// TIA Portal V20 export
FUNCTION_BLOCK "FB_WarmUP"   // FB530, SCL
{ S7_Optimized_Access := 'TRUE' }
// stored: AutoNumber false, MemoryReserve 100, SetENOAutomatically false
   VAR
      sWarmUpTimer : Time;
      sLimitedWarmupTime : Bool;
      sUnlimitedWarmupTime : Bool;
      sActualWarmupTime : Time;
      sRemainingWarmupMinutes : Int;
      sDeltaTimeWarmup : Time;
      sLimitedWarmUP : TON_TIME;
      sStartWarmup { S7_SetPoint := 'True'} : Bool;
      sUnlimitedWarmUP : TON_TIME;
      sUnlimitedWarmUPCounter { S7_SetPoint := 'True'} : "FB_TimeCounter";
   END_VAR
   VAR CONSTANT
      WU_MIN : Int := 30;
   END_VAR
BEGIN
   REGION Description header 
       //==================================================================================
       // POSALUX Swiss SA / (C) Copyright 2024
       //----------------------------------------------------------------------------------
       // Title: Laser Warm-up
       // Comment/Function: 
       // This block manages the laser warm-up process. It includes functionality for both limited
       // and unlimited warm-up times.
       //
       // Author: [Gowsigan SRITHARAN]
       // Engineering: TIA Portal [version]
       //----------------------------------------------------------------------------------
       // Change log table:
       // Version  | Date     | Expert in charge | Changes applied
       // ---------|----------|------------------|------------------------------------
       // 00.00.01 | 20250224 | gsr              | First released version
       // 00.00.02 | 20250314 | wfa              | Modification unlimited timer
       // ==================================================================================
   END_REGION

   REGION Selection Warm-UP mode: limited or unlimited
       // Timer for unlimited Warm-UP detection
       #sUnlimitedWarmUP(IN := "DB_McpKeyboardSignals".sK14_WarmUp.sKeySWStatus OR "DB_HmiKeyboardSignals".sK14_WarmUp.sKeySWStatus,
                         PT := T#2s);

       // Warm-up mode selection logic
       IF ("DB_McpKeyboardSignals".sK14_WarmUp.sKeySWStatus OR "DB_HmiKeyboardSignals".sK14_WarmUp.sKeySWStatus) AND "LBP_ModeGroup".E_AUTO AND NOT #sUnlimitedWarmUP.Q THEN
           // Activate unlimited Warm-UP when key is initially pressed
           #sLimitedWarmupTime := FALSE;
           #sUnlimitedWarmupTime := TRUE;
           #sStartWarmup := TRUE;
       ELSIF "DB_McpKeyboardSignals".sK14_WarmUp.sKeySWStatus AND "DB_HmiKeyboardSignals".sK14_WarmUp.sKeySWStatus AND "LBP_ModeGroup".E_AUTO AND #sUnlimitedWarmUP.Q THEN
           // Switch to limited Warm-UP if key is held for 2 seconds
           #sLimitedWarmupTime := TRUE;
           #sUnlimitedWarmupTime := FALSE;
           #sStartWarmup := TRUE;
           #sWarmUpTimer := DINT_TO_TIME(DINT_TO_INT(#WU_MIN * 60 * 1000)); // Limited time in milliseconds
       ELSIF "DB_McpKeyboardSignals".sK14_WarmUp.sKeySWToggleStatus = FALSE AND "DB_HmiKeyboardSignals".sK14_WarmUp.sKeySWToggleStatus THEN
           #sLimitedWarmupTime := FALSE;
           #sUnlimitedWarmupTime := FALSE;
           #sStartWarmup := FALSE;
       END_IF;
   END_REGION

   REGION Warm-UP Counter (Unlimited Warm-Up)
       #sUnlimitedWarmUPCounter(iStart := #sUnlimitedWarmupTime AND ("LBP_Chan1".E_ProgRunning OR "LBP_Chan1".E_ProgWait OR "LBP_Chan1".E_ProgStop),
                                iReset := NOT "DB_McpKeyboardSignals".sK14_WarmUp.sKeySWToggleStatus AND NOT "DB_HmiKeyboardSignals".sK14_WarmUp.sKeySWToggleStatus);
   END_REGION ;

   REGION Warm-UP Timer  (Limited Warm-up)  
       // Start the Warm-UP timer
       #sLimitedWarmUP.TON(IN := #sLimitedWarmupTime AND ("LBP_Chan1".E_ProgRunning OR "LBP_Chan1".E_ProgWait OR "LBP_Chan1".E_ProgStop),
                           PT := #sWarmUpTimer);

       IF #sLimitedWarmUP.Q THEN
           "DB_McpKeyboardSignals".sK14_WarmUp.sKeySWToggleStatus := FALSE;
           "DB_HmiKeyboardSignals".sK14_WarmUp.sKeySWToggleStatus := FALSE;
       END_IF;
   END_REGION

   REGION Update NC inputs and MCP LED status
       "LBP_NC".A_Set_Inp34 := "DB_McpKeyboardSignals".sK14_WarmUp.sKeySWToggleStatus OR "DB_HmiKeyboardSignals".sK14_WarmUp.sKeySWToggleStatus;

       "DB_McpKeyboardSignals".sK14_WarmUp.sLedSWStatus :=
       "DB_McpKeyboardSignals".sK14_WarmUp.sKeySWToggleStatus
       AND (#sUnlimitedWarmupTime OR "Clock_2Hz");

       "DB_HmiKeyboardSignals".sK14_WarmUp.sLedSWStatus :=
       "DB_HmiKeyboardSignals".sK14_WarmUp.sKeySWToggleStatus
       AND (#sUnlimitedWarmupTime OR "Clock_2Hz");
   END_REGION

   REGION Display Remaining Time
       IF #sLimitedWarmupTime THEN
           // Display remaining time for limited warm-up
           "DB_HMIStatus".WarmUpTime := DINT_TO_REAL(TIME_TO_DINT(#sLimitedWarmUP.PT - #sLimitedWarmUP.ET)) / 1000.0;
       ELSIF #sUnlimitedWarmupTime THEN
           // Display elapsed time for unlimited warm-up
           "DB_HMIStatus".WarmUpTime := #sUnlimitedWarmUPCounter.ioSecondsCumul;
       ELSE
           // Reset display when conditions are not met
           "DB_HMIStatus".WarmUpTime := 0;
       END_IF;
   END_REGION

   REGION Warm-UP Message
       IF "LBP_ModeGroup".E_AUTO AND "LBP_NC".A_Set_Inp34 AND
           ("LBP_Chan1".E_ProgRunning OR "LBP_Chan1".E_ProgWait OR "LBP_Chan1".E_ProgStop) THEN
           "LBP_AlarmMsgs".UserA[0].A70UUxx[35] := TRUE;
       END_IF;
   END_REGION

   REGION Warm-UP Status
       "DB_HMIStatus".WarmUpOn := #sStartWarmup;
   END_REGION

   REGION Warm-UP Status To NC
       "DB_PLC_ISO_IHM".WarmUpOn := "DB_McpKeyboardSignals".sK14_WarmUp.sKeySWToggleStatus OR "DB_HmiKeyboardSignals".sK14_WarmUp.sKeySWToggleStatus;
   END_REGION
END_FUNCTION_BLOCK
